(* PLC project Blank Project, Blank Blank 1.0 *)
(* stored: creationDateTime 2016-05-18T21:14:07, modificationDateTime 2016-11-26T20:38:26 *)

PROGRAM My_Program
  VAR
    transformer AT %QX0.0 : BOOL := 1;
    switch1 AT %QW0 : INT := 1;
  END_VAR
  VAR
    switch2 AT %QW1 : INT := 1;
  END_VAR
  VAR
    TON0 : TON;
    TON1 : TON;
  END_VAR

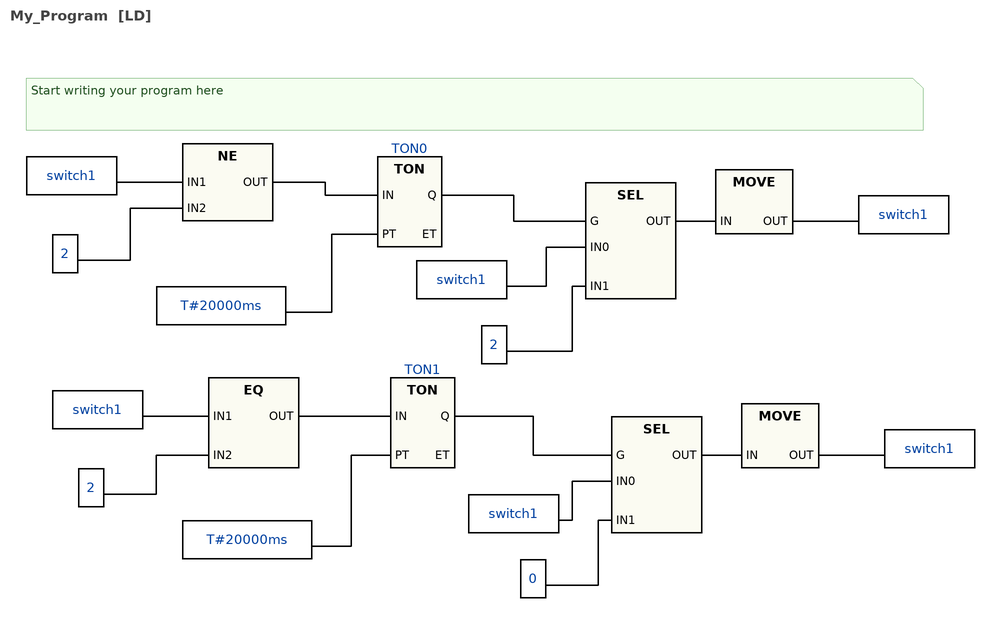
(* LD diagram, written out as Structured Text *)
(* Start writing your program here *)
TON0(IN := switch1 <> 2, PT := T#20000ms);
switch1 := SEL(TON0.Q, switch1, 2);
TON1(IN := switch1 = 2, PT := T#20000ms);
switch1 := SEL(TON1.Q, switch1, 0);
END_PROGRAM

CONFIGURATION Config0
  RESOURCE Res0 ON PLC
    TASK TaskMain(INTERVAL := T#50ms, PRIORITY := 0);
    PROGRAM Inst0 WITH TaskMain : My_Program;
  END_RESOURCE
END_CONFIGURATION
